// TIA Portal V19 export
DATA_BLOCK "Rollformer_PERS"   // DB126
// stored: MemoryReserve 100
   VAR RETAIN
      PersistentValues : "udt_Rollformer_Pers";
   END_VAR
BEGIN
   PersistentValues.Machine.Par.ExtraLow_Enable := FALSE;
   PersistentValues.Machine.Par.ExtraLow_VelPercentage := 10.0;
   PersistentValues.Feed.Par.PosTolerance := 0.1;
   PersistentValues.Feed.Par.DelayInPosition := T#0MS;
   PersistentValues.Feed.Par.Man.VelBwd := 5000.0;
   PersistentValues.Feed.Par.Man.VelFwdHigh := 5000.0;
   PersistentValues.Feed.Par.Man.VelFwdLow := 5000.0;
   PersistentValues.Feed.Par.Man.Acc := 500.0;
   PersistentValues.Feed.Par.Man.Dec := 500.0;
   PersistentValues.Feed.Par.Man.Jerk := 5000.0;
   PersistentValues.Feed.Par.Man.DelayChangeVel := T#5S;
   PersistentValues.Feed.Par.Man.UsePositionControl := FALSE;
   PersistentValues.Feed.Pers_Data.AxisEncoderSelection_OK := TRUE;
   PersistentValues.Feed.Pers_Data.AxisParameters_OK := TRUE;
   PersistentValues.Feed.Pers_Data.AxisReloadPostion_OK := TRUE;
   PersistentValues.Feed.Pers_Data.ActualPosition := 647863.802;
END_DATA_BLOCK
